PROGRAM PRG_Main
VAR
	bTestInput: BOOL;
	bTestOutput: BOOL;
	fbMachine: FB_ExampleMachine;
	fbStation1: FB_ExampleStation;
	fbStation2: FB_ExampleStation;
	fbStation3: FB_ExampleStation;
	fbStation4: FB_ExampleStation;
	bStart: BOOL;
	bAbort: BOOL;
	bReset: BOOL;
	bStop: BOOL;
	bSuspend: BOOL;
	fbDevice1: FB_ExampleDevice;
	fbDevice2: FB_ExampleDevice;
	fbDevice3: FB_ExampleDevice;
	fbDevice4: FB_ExampleDevice;
	bPoweredOn: BOOL;
//	FB_AdsDeviceAPI_0: FB_AdsDeviceAPI;
	FB_AdsDeviceAPI_0 : FB_AdsCommandRouter;
	MyLaser1: FB_KeyenceLaserMarkerMDX2000;
	bConnectToLaserMarker: BOOL;
	bRes_LaserConnected: BOOL;
	bTestADSServer: BOOL;
	strTarget: T_MaxString;
	strCommand: T_MaxString;
	arrParams: T_ApiMethodParameters;
	MyResults: T_MaxString;
	bInterfaceTest : BOOL;
	temp: BOOL;
	bDisconnectFromLaserMarker: BOOL;
	bRes_LaserDisconnected: BOOL;
	bPeakCurrentProgramInLaser: BOOL;
	bRes_PeakCurrentProgramInLaser: BOOL;
	bSendProgramToLaser: BOOL;
	bRes_SendProgramtoLaser: BOOL;
	filepath : STRING;
	LaserMemoryLocation : INT;
END_VAR

bTestOutput := bTestInput;

A_Machine();
//A_Station1();
//A_Station2();
//A_Station3();
//A_Station4();
//bInterfaceTest := MyLaser1.fbApi.P_bDeviceInterfaceBusy;
IF bConnectToLaserMarker THEN
	bRes_LaserConnected := MyLaser1.M_Connect();
//	IF bRes_LaserConnected THEN
//	//Add some timer based logic to do error handling.
//		bConnectToLaserMarker := FALSE;
//	END_IF
	bConnectToLaserMarker := FALSE;
END_IF
IF bRes_LaserConnected THEN
	//Add some timer based logic to do error handling.
//		bConnectToLaserMarker := FALSE;
END_IF

//IF bDisconnectFromLaserMarker THEN
//	bRes_LaserDisconnected := MyLaser1.M_Disconnect();
//	bDisconnectFromLaserMarker := FALSE;
//END_IF
//IF bRes_LaserDisconnected THEN
////		bDisconnectFromLaserMarker := FALSE;
//END_IF

//IF bPeakCurrentProgramInLaser THEN
//	bRes_PeakCurrentProgramInLaser := MyLaser1.M_PeakCurrentProgram();
//	bPeakCurrentProgramInLaser := FALSE;
//END_IF

//IF bRes_PeakCurrentProgramInLaser THEN
////		bPeakCurrentProgramInLaser := FALSE;
//END_IF

//IF bSendProgramToLaser THEN
//	bRes_SendProgramtoLaser := MyLaser1.M_SendProgramtoLaser(filepath,LaserMemoryLocation);
//	bSendProgramToLaser := FALSE;
////	IF bRes_SendProgramtoLaser THEN
////		bSendProgramToLaser := FALSE;
////	END_IF
//END_IF

//IF bRes_SendProgramtoLaser THEN
//		bSendProgramToLaser := FALSE;
//END_IF

ACTION A_Machine:
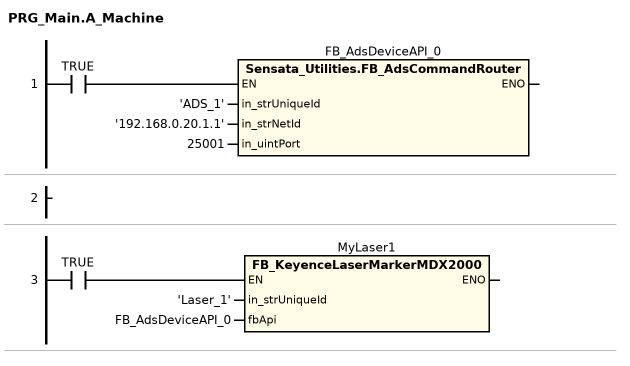
// NETWORK 1
FB_AdsDeviceAPI_0(in_strUniqueId := 'ADS_1', in_strNetId := '192.168.0.20.1.1', in_uintPort := 25001); // Sensata_Utilities.FB_AdsCommandRouter

// NETWORK 2

// NETWORK 3
MyLaser1(in_strUniqueId := 'Laser_1', fbApi := FB_AdsDeviceAPI_0); // FB_KeyenceLaserMarkerMDX2000
END_ACTION

ACTION A_Station1:
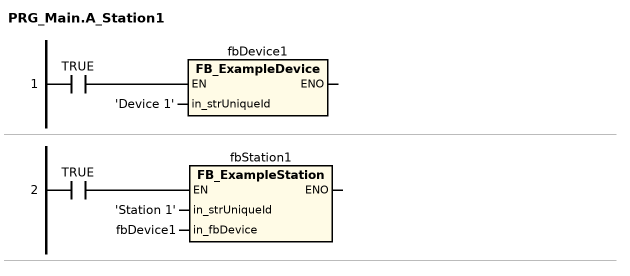
// NETWORK 1
fbDevice1(in_strUniqueId := 'Device 1'); // FB_ExampleDevice

// NETWORK 2
fbStation1(in_strUniqueId := 'Station 1', in_fbDevice := fbDevice1); // FB_ExampleStation
END_ACTION

ACTION A_Station2:
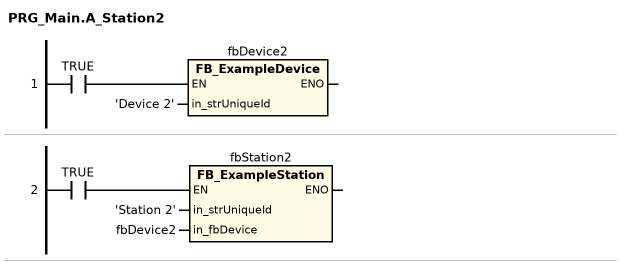
// NETWORK 1
fbDevice2(in_strUniqueId := 'Device 2'); // FB_ExampleDevice

// NETWORK 2
fbStation2(in_strUniqueId := 'Station 2', in_fbDevice := fbDevice2); // FB_ExampleStation
END_ACTION

ACTION A_Station3:
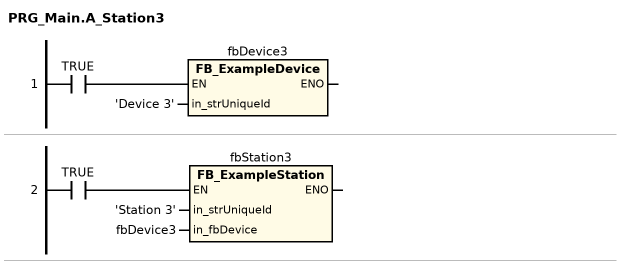
// NETWORK 1
fbDevice3(in_strUniqueId := 'Device 3'); // FB_ExampleDevice

// NETWORK 2
fbStation3(in_strUniqueId := 'Station 3', in_fbDevice := fbDevice3); // FB_ExampleStation
END_ACTION

ACTION A_Station4:
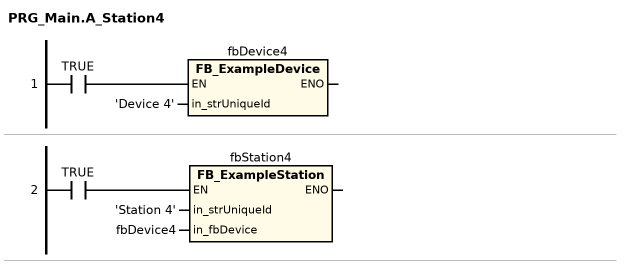
// NETWORK 1
fbDevice4(in_strUniqueId := 'Device 4'); // FB_ExampleDevice

// NETWORK 2
fbStation4(in_strUniqueId := 'Station 4', in_fbDevice := fbDevice4); // FB_ExampleStation
END_ACTION

END_PROGRAM

(* stored: Version 1.1.0.1, ProductVersion 3.1.4024.11
   POU PRG_Main: Id {b13f0be3-4c97-4edc-94e2-8c6f67cb8665}, SpecialFunc None
   Action A_Machine: Id {f2ef6f5c-8a40-4c62-8311-b3186050d362}
   Action A_Station1: Id {504119fa-b0a8-489a-9a37-499472501127}
   Action A_Station2: Id {21ea2e05-12d0-4cac-a384-2d35f55a53ab}
   Action A_Station3: Id {a8c1dd1b-134a-4dcf-b99f-4a08bcf13697}
   Action A_Station4: Id {f4929fa8-ed63-4a91-b73a-b4250062275b} *)
